// TIA Portal V16 export
// export: Created 2021-09-08T12:46:14.932706Z, ExportSetting WithDefaults, DisplayName Totally Integrated Automation Portal, DisplayVersion V16 Update 3, DisplayName TIA Portal Version Control Interface, DisplayVersion V16 Update 2, DisplayName TIA Portal Openness, DisplayVersion V16 Update 3, DisplayName TIA Portal Teamcenter Gateway, DisplayVersion V16, DisplayName STEP 7 Professional, DisplayVersion V16 Update 3, DisplayName STEP 7 Safety, DisplayVersion V16, DisplayName WinCC Advanced, DisplayVersion V16 Update 3
DATA_BLOCK "AllUF_DB"   // DB28
VERSION : 0.1
// stored: AutoNumber true, DBAccessibleFromOPCUA true, InstanceOfName AllUF, InstanceOfType FB
"AllUF"
   // VAR
   //    reqNumbWorkUF { ExternalVisible := 'False'; ExternalWritable := 'False'} : USInt;
   //    readyUF : Array[0..1] of Bool;
   //    workUF : Array[0..1] of Bool;
   //    cmUF : Array[0..1] of Bool;
   //    HandlerUF1 { S7_SetPoint := 'True'} : "HandlerUF";
   //    HandlerUF2 { S7_SetPoint := 'True'} : "HandlerUF";
   // END_VAR
BEGIN
END_DATA_BLOCK
